% RSLogix 500 project Ventura 3d crap.RSS, saved by version 11.00.00.00 %
PROJECT "UNTITLED"    % processor: MicroLogix 1400 %

PROGRAM FILES
  LAD 2   31 rungs

DATA FILES
  O0 OUTPUT  6 elements
  I1 INPUT  15 elements
  S2 STATUS  66 elements
  B3 BINARY  10 elements
  T4 TIMER  12 elements
  C5 COUNTER  2 elements
  R6 CONTROL  1 elements
  N7 INTEGER  15 elements
  F8 FLOAT  3 elements

LADDER 2
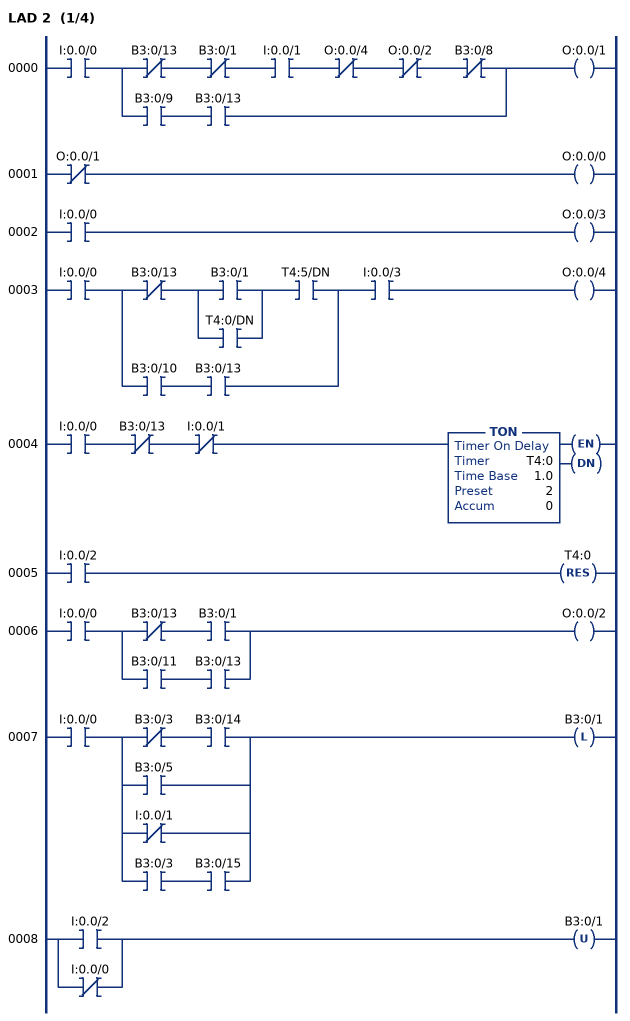
% Rung: 0 %
SOR XIC I:0.0/0 BST XIO B3:0/13 XIO B3:0/1 XIC I:0.0/1 XIO O:0.0/4 XIO O:0.0/2 XIO B3:0/8 NXB XIC B3:0/9 XIC B3:0/13 BND OTE O:0.0/1 EOR
% Rung: 1 %
SOR XIO O:0.0/1 OTE O:0.0/0 EOR
% Rung: 2 %
SOR XIC I:0.0/0 OTE O:0.0/3 EOR
% Rung: 3 %
SOR XIC I:0.0/0 BST XIO B3:0/13 BST XIC B3:0/1 NXB XIC T4:0/DN BND XIC T4:5/DN NXB XIC B3:0/10 XIC B3:0/13 BND XIC I:0.0/3 OTE O:0.0/4 EOR
% Rung: 4 %
SOR XIC I:0.0/0 XIO B3:0/13 XIO I:0.0/1 TON T4:0 1.0 2 0 EOR
% Rung: 5 %
SOR XIC I:0.0/2 RES T4:0 EOR
% Rung: 6 %
SOR XIC I:0.0/0 BST XIO B3:0/13 XIC B3:0/1 NXB XIC B3:0/11 XIC B3:0/13 BND OTE O:0.0/2 EOR
% Rung: 7 %
SOR XIC I:0.0/0 BST XIO B3:0/3 XIC B3:0/14 NXB BST XIC B3:0/5 NXB BST XIO I:0.0/1 NXB XIC B3:0/3 XIC B3:0/15 BND BND BND OTL B3:0/1 EOR
% Rung: 8 %
SOR BST XIC I:0.0/2 NXB XIO I:0.0/0 BND OTU B3:0/1 EOR

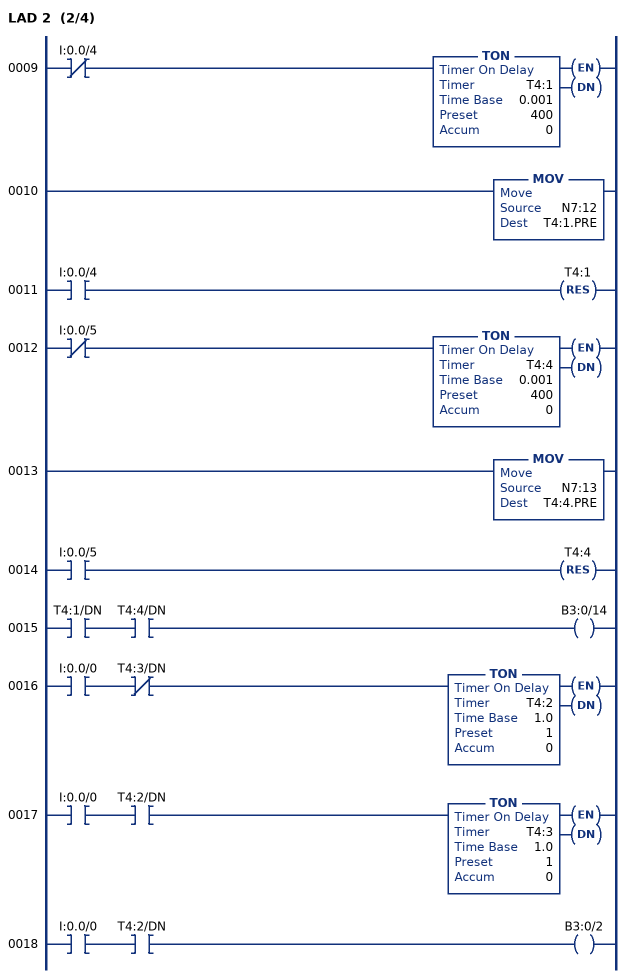
% Rung: 9 %
SOR XIO I:0.0/4 TON T4:1 0.001 400 0 EOR
% Rung: 10 %
SOR MOV N7:12 T4:1.PRE EOR
% Rung: 11 %
SOR XIC I:0.0/4 RES T4:1 EOR
% Rung: 12 %
SOR XIO I:0.0/5 TON T4:4 0.001 400 0 EOR
% Rung: 13 %
SOR MOV N7:13 T4:4.PRE EOR
% Rung: 14 %
SOR XIC I:0.0/5 RES T4:4 EOR
% Rung: 15 %
SOR XIC T4:1/DN XIC T4:4/DN OTE B3:0/14 EOR
% Rung: 16 %
SOR XIC I:0.0/0 XIO T4:3/DN TON T4:2 1.0 1 0 EOR
% Rung: 17 %
SOR XIC I:0.0/0 XIC T4:2/DN TON T4:3 1.0 1 0 EOR
% Rung: 18 %
SOR XIC I:0.0/0 XIC T4:2/DN OTE B3:0/2 EOR

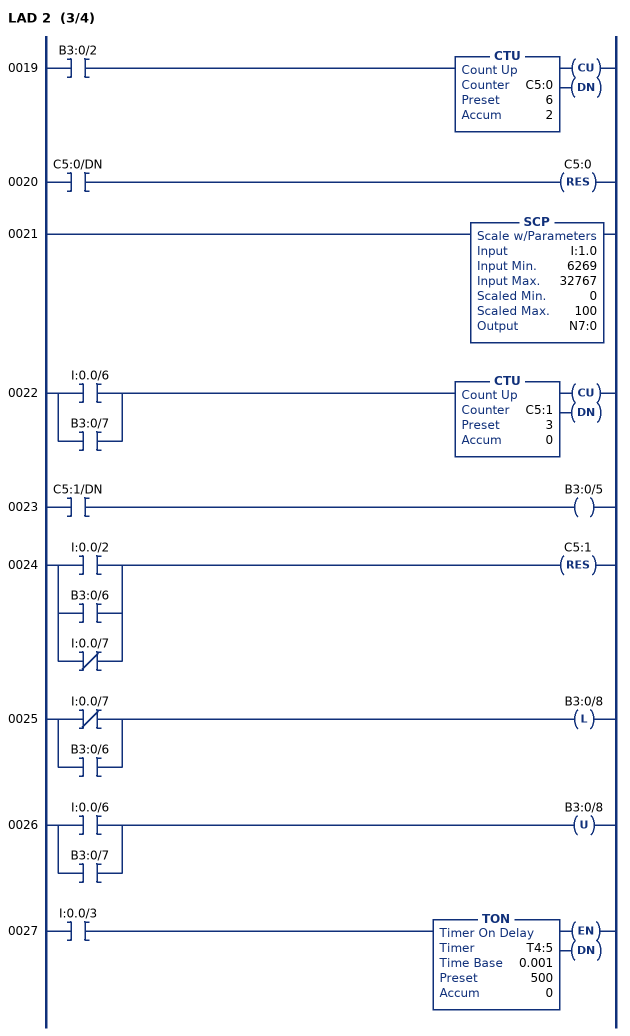
% Rung: 19 %
SOR XIC B3:0/2 CTU C5:0 6 2 EOR
% Rung: 20 %
SOR XIC C5:0/DN RES C5:0 EOR
% Rung: 21 %
SOR SCP I:1.0 6269 32767 0 100 N7:0 EOR
% Rung: 22 %
SOR BST XIC I:0.0/6 NXB XIC B3:0/7 BND CTU C5:1 3 0 EOR
% Rung: 23 %
SOR XIC C5:1/DN OTE B3:0/5 EOR
% Rung: 24 %
SOR BST XIC I:0.0/2 NXB BST XIC B3:0/6 NXB XIO I:0.0/7 BND BND RES C5:1 EOR
% Rung: 25 %
SOR BST XIO I:0.0/7 NXB XIC B3:0/6 BND OTL B3:0/8 EOR
% Rung: 26 %
SOR BST XIC I:0.0/6 NXB XIC B3:0/7 BND OTU B3:0/8 EOR
% Rung: 27 %
SOR XIC I:0.0/3 TON T4:5 0.001 500 0 EOR

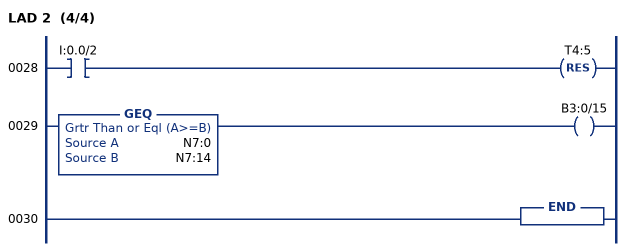
% Rung: 28 %
SOR XIC I:0.0/2 RES T4:5 EOR
% Rung: 29 %
SOR GEQ N7:0 N7:14 OTE B3:0/15 EOR
% Rung: 30 %
SOR END EOR

DATA TABLE (non-zero values as saved)
DATA B3
% B3:0 % 0X0108 0X000B 0X0000 0X0000 0X0000 0X0000 0X0000 0X0000 0X0000 0X0001
DATA T4
% .PRE .ACC %
% T4:0 % 2 0
% T4:1 % 400 0
% T4:2 % 1 0
% T4:3 % 1 0
% T4:4 % 400 0
% T4:5 % 500 0
% T4:6 % 1440 1530
% T4:10 % 6 4
% T4:11 % 5 0
DATA C5
% .PRE .ACC %
% C5:0 % 6 2
% C5:1 % 3 0
DATA N7
% N7:0 % 8 51 51 51 51 52 102 153 204 256
% N7:10 % 51 1470 400 400 75
DATA F8
% F8:0 % 0 22161 86.55965
